TYPE eHomeModeOption :
(
	eNEGATIVE := 0 ,
	ePOSITIVE := 1
);
END_TYPE

(* stored: Version 1.1.0.1, ProductVersion 3.1.4024.3
   DUT eHomeModeOption: Id {ff6e8c68-e25a-0fad-2a0e-5c850ca11a64} *)
